FUNCTION_BLOCK FB_Maintenance IMPLEMENTS I_State
VAR_INPUT
	(* Pointer to the ATM Machine*)
	pATM_Machine	: POINTER TO FB_ATM_Machine;
END_VAR
VAR_OUTPUT
END_VAR
VAR
END_VAR

METHOD Cancel : BOOL
END_METHOD

METHOD Card_Ejected : BOOL
END_METHOD

METHOD Card_Inserted : BOOL
END_METHOD

PROPERTY Description : E_StateDescription
GET
Description := E_StateDescription.Maintenance;
END_GET
END_PROPERTY

METHOD Failure : BOOL
END_METHOD

METHOD FB_Init : BOOL
VAR_INPUT
	(* if TRUE, the retain variables are initialized (warm start / cold start)*)
	bInitRetains	: BOOL;
	(* if TRUE, the instance afterwards gets moved into the copy code (online change)*)
	bInCopyCode	: BOOL;
	(* Pointer to the ATM Machine*)
	pATM_Machine	: POINTER TO FB_ATM_Machine;
END_VAR
THIS^.pATM_Machine := pATM_Machine;
END_METHOD

METHOD Op : BOOL
ADSLOGSTR(ADSLOG_MSGTYPE_LOG, 'Exiting Service mode, going to self test', '');
pATM_Machine^.SetState(pATM_Machine^.SelfTestState);
END_METHOD

METHOD Service : BOOL
END_METHOD

METHOD SystemTest_OK : BOOL
END_METHOD

METHOD Turn_Off : BOOL
END_METHOD

METHOD Turn_On : BOOL
END_METHOD

END_FUNCTION_BLOCK

(* stored: Version 1.1.0.1, ProductVersion 3.1.4024.12
   POU FB_Maintenance: Id {422bee07-fab0-086f-2f20-2f473840af98}, SpecialFunc None
   Method Cancel: Id {fc6c514b-2a24-0485-0094-7f9672024860}
   Method Card_Ejected: Id {f0c20272-59ca-04aa-17cf-f0dc9b6e6caa}
   Method Card_Inserted: Id {8c8901b8-6177-09cf-0171-70900555bba1}
   Property Description: Id {9563a445-e11a-0e6c-0c59-44fdd0b4d03f}
   Get Get: Id {f4aa627d-a63a-0b8c-16ea-3a081815301d}
   Method Failure: Id {5c7b77fb-733d-070b-292d-1bd3ac175be9}
   Method FB_Init: Id {724c03c1-3a42-00fb-371d-203832591578}
   Method Op: Id {d5b1852a-c23d-0073-23f0-eda99df56713}
   Method Service: Id {5643db20-9040-00ed-10c1-8d0666a21e31}
   Method SystemTest_OK: Id {e4e24f0f-5074-0c16-0c9d-ff973e36ac56}
   Method Turn_Off: Id {904c14f7-b1ec-0e92-0ab3-92a000c17c86}
   Method Turn_On: Id {77c37fbd-c644-01ab-24b8-e342a38b3aae} *)
